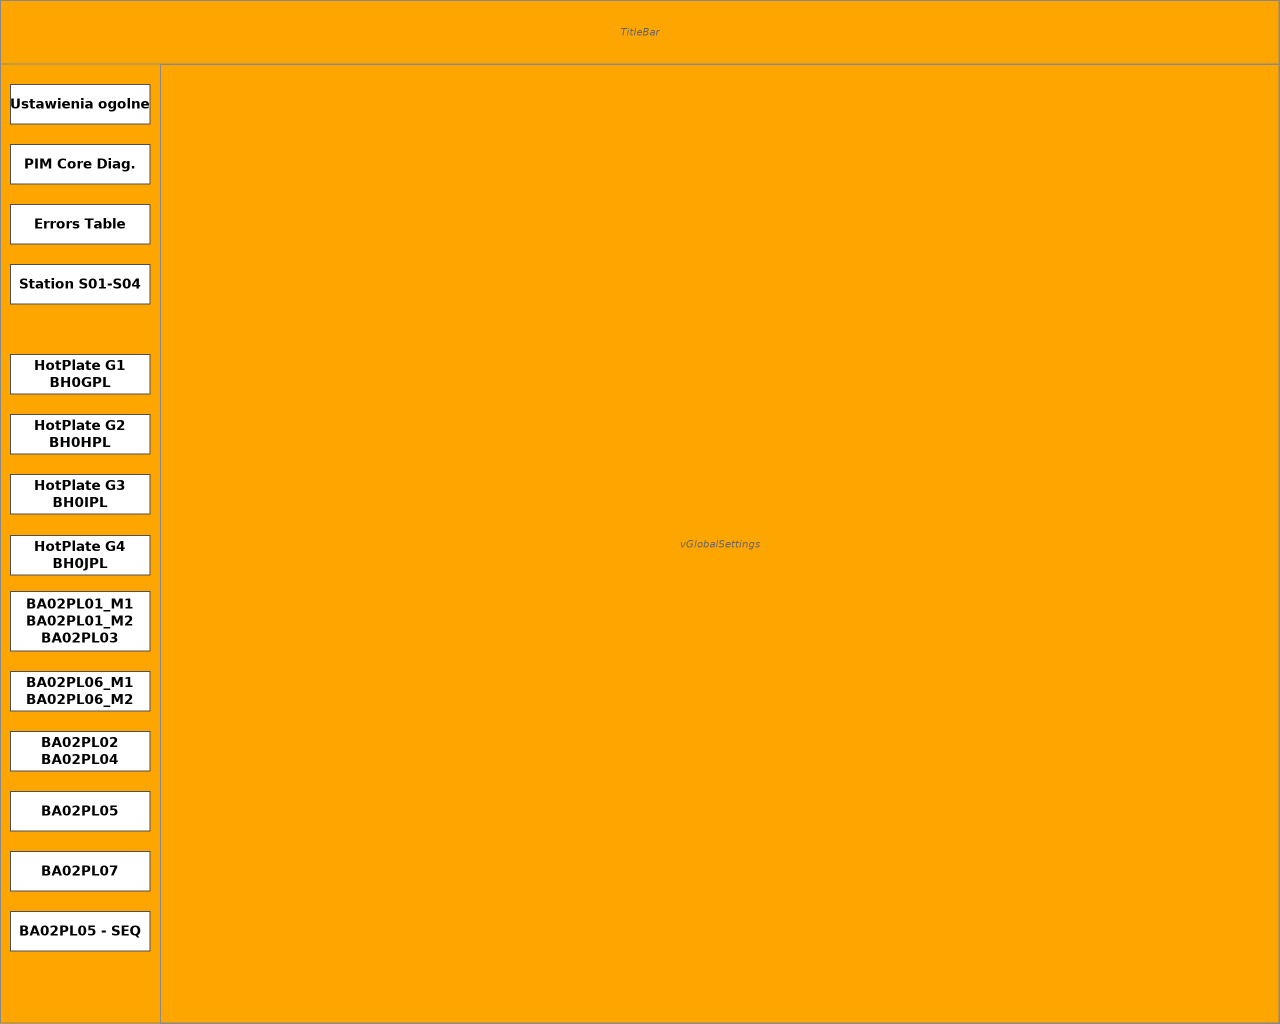
VISUALIZATION HomeVisu  // 1280x1024
    Rectangle (10,264 140x40), "Station S01-S04"
        OnMouseClick: FrameSelectionChange Selection=SelectedFrame=2d0b6361-e960-4000-ab6f-31a4b2a9c614, Selection=3, GlobSel=AssignType=Directly, SelType=Locally
    Frame (160,64 1120x960)
        shows vGlobalSettings()
        shows vErrorsData()
        shows AircomLibrary.vSQL_CoreDiag(fbData := GVL.fbSqlCore)
        shows vS01_04()
        shows vHP3_MainSet(fbHP_M1 := MAIN.fbHotPlate_G1_M1, fbHP_M2 := MAIN.fbHotPlate_G1_M2, fbHP_M3 := MAIN.fbHotPlate_G1_M3, NestNumber := 1, sSocketName := 'BH0GPL')
        shows vHP3_MainSet(fbHP_M1 := MAIN.fbHotPlate_G2_M1, fbHP_M2 := MAIN.fbHotPlate_G2_M2, fbHP_M3 := MAIN.fbHotPlate_G2_M3, NestNumber := 2, sSocketName := 'BH0HPL')
        shows vHP3_MainSet(fbHP_M1 := MAIN.fbHotPlate_G3_M1, fbHP_M2 := MAIN.fbHotPlate_G3_M2, fbHP_M3 := MAIN.fbHotPlate_G3_M3, NestNumber := 3, sSocketName := 'BH0IPL')
        shows vFrameFillingLine_1()
        shows vFrameFillingLine_2()
        shows vUnderPressureFrame()
        shows vDetectionTunelFrame(stInOuts := GVL_IO.stTunelInOuts, stParams := GVL.st_Tunel_Params, iWorkStep := MAIN.fb_Tunel_Machine.iWorkStep)
        shows vTransporterSequence(iWorkStep := MAIN.fbTransporterUnderpressure.iWorkStep)
        shows vHP3_MainSet(fbHP_M1 := MAIN.fbHotPlate_G4_M1, fbHP_M2 := MAIN.fbHotPlate_G4_M2, fbHP_M3 := MAIN.fbHotPlate_G4_M3, NestNumber := 4, sSocketName := 'BH0JPL')
        shows vStations19_21_22()
        [6]: fbData=MAIN.fbLL19_2_EOL_Chamber_II, Settings=GVL.stLL19_EOL_Chamber_2_Settings, Name='Right chamber'
        p2683556743: GVL.stLJ20_DTL_WorkParams
        p1709583229: GVL.stLL19_EOL_Settings_I
        p2719655782: MAIN.fbLL19_2_EOL3
        p3094409976: GVL.stLL19_EOL_Settings_II
        p74549115: 'Left chamber'
        p3369830373: 'Right chamber'
        p4001053958: MAIN.fbLN21_DetectionTunel
        p2893311244: GVL.stLN21_DTL_WorkParams
        p3191039994: MAIN.stStacjaC03PL21
    Frame (0,0 1280x64)
        shows TitleBar()
    Rectangle (10,84 140x40), "Ustawienia ogolne"
        OnMouseClick: FrameSelectionChange Selection=SelectedFrame=2d0b6361-e960-4000-ab6f-31a4b2a9c614, GlobSel=AssignType=Directly, SelType=Locally
    Rectangle (10,204 140x40), "Errors Table"
        OnMouseClick: FrameSelectionChange Selection=SelectedFrame=2d0b6361-e960-4000-ab6f-31a4b2a9c614, Selection=1, GlobSel=AssignType=Directly, SelType=Locally
    Rectangle (10,144 140x40), "PIM Core Diag."
        OnMouseClick: FrameSelectionChange Selection=SelectedFrame=2d0b6361-e960-4000-ab6f-31a4b2a9c614, Selection=2, GlobSel=AssignType=Directly, SelType=Locally
    Rectangle (10,354 140x40), "HotPlate G1 BH0GPL"
        OnMouseClick: FrameSelectionChange Selection=SelectedFrame=2d0b6361-e960-4000-ab6f-31a4b2a9c614, Selection=4, GlobSel=AssignType=Directly, SelType=Locally
    Rectangle (10,414 140x40), "HotPlate G2 BH0HPL"
        OnMouseClick: FrameSelectionChange Selection=SelectedFrame=2d0b6361-e960-4000-ab6f-31a4b2a9c614, Selection=5, GlobSel=AssignType=Directly, SelType=Locally
    Rectangle (10,474 140x40), "HotPlate G3 BH0IPL"
        OnMouseClick: FrameSelectionChange Selection=SelectedFrame=2d0b6361-e960-4000-ab6f-31a4b2a9c614, Selection=6, GlobSel=AssignType=Directly, SelType=Locally
    Rectangle (10,591 140x60), "BA02PL01_M1 BA02PL01_M2 BA02PL03"
        OnMouseClick: FrameSelectionChange Selection=SelectedFrame=2d0b6361-e960-4000-ab6f-31a4b2a9c614, Selection=7, GlobSel=AssignType=Directly, SelType=Locally
    Rectangle (10,671 140x40), "BA02PL06_M1 BA02PL06_M2"
        OnMouseClick: FrameSelectionChange Selection=SelectedFrame=2d0b6361-e960-4000-ab6f-31a4b2a9c614, Selection=8, GlobSel=AssignType=Directly, SelType=Locally
    Rectangle (10,731 140x40), "BA02PL02 BA02PL04"
        OnMouseClick: FrameSelectionChange Selection=SelectedFrame=2d0b6361-e960-4000-ab6f-31a4b2a9c614, Selection=8, GlobSel=AssignType=Directly, SelType=Locally
    Rectangle (10,791 140x40), "BA02PL05"
        OnMouseClick: FrameSelectionChange Selection=SelectedFrame=2d0b6361-e960-4000-ab6f-31a4b2a9c614, Selection=9, GlobSel=AssignType=Directly, SelType=Locally
    Rectangle (10,851 140x40), "BA02PL07"
        OnMouseClick: FrameSelectionChange Selection=SelectedFrame=2d0b6361-e960-4000-ab6f-31a4b2a9c614, Selection=10, GlobSel=AssignType=Directly, SelType=Locally
    Rectangle (10,911 140x40), "BA02PL05 - SEQ"
        OnMouseClick: FrameSelectionChange Selection=SelectedFrame=2d0b6361-e960-4000-ab6f-31a4b2a9c614, Selection=11, GlobSel=AssignType=Directly, SelType=Locally
    Rectangle (10,535 140x40), "HotPlate G4 BH0JPL"
        OnMouseClick: FrameSelectionChange Selection=SelectedFrame=2d0b6361-e960-4000-ab6f-31a4b2a9c614, Selection=12, GlobSel=AssignType=Directly, SelType=Locally
END_VISUALIZATION

(* stored: Version 1.1.0.1, ProductVersion 3.1.4024.13
   Visu HomeVisu: Id {8eb58b9b-fbaf-48d4-8013-9086807328f0} *)
